// Mitsubishi GX Works2 project: plc_torque1   PLC: FX3U/FX3UC

PROGRAM MAIN
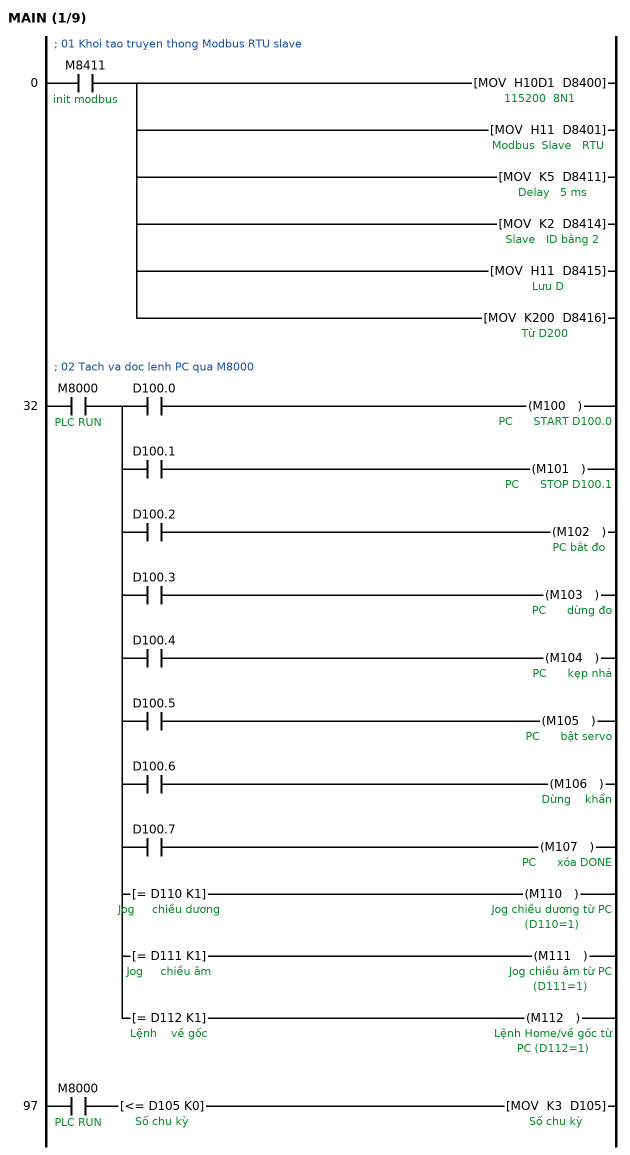
; 01 Khoi tao truyen thong Modbus RTU slave
0     LD      M8411  ; init modbus
      MOV     H10D1 D8400  ; 115200  8N1
      MOV     H11 D8401  ; Modbus  Slave   RTU
      MOV     K5 D8411  ; Delay   5 ms
      MOV     K2 D8414  ; Slave   ID bằng 2
      MOV     H11 D8415  ; Lưu D
      MOV     K200 D8416  ; Từ D200
; 02 Tach va doc lenh PC qua M8000
32    LD      M8000  ; PLC RUN
      MPS
      AND     D100.0
      OUT     M100  ; PC      START D100.0
      MRD
      AND     D100.1
      OUT     M101  ; PC      STOP D100.1
      MRD
      AND     D100.2
      OUT     M102  ; PC bắt đo
      MRD
      AND     D100.3
      OUT     M103  ; PC      dừng đo
      MRD
      AND     D100.4
      OUT     M104  ; PC      kẹp nhả
      MRD
      AND     D100.5
      OUT     M105  ; PC      bật servo
      MRD
      AND     D100.6
      OUT     M106  ; Dừng    khẩn
      MRD
      AND     D100.7
      OUT     M107  ; PC      xóa DONE
      MRD
      LD=     D110 K1  ; Jog     chiều dương
      ANB
      OUT     M110  ; Jog chiều dương từ PC (D110=1)
      MRD
      LD=     D111 K1  ; Jog     chiều âm
      ANB
      OUT     M111  ; Jog chiều âm từ PC (D111=1)
      MPP
      LD=     D112 K1  ; Lệnh    về gốc
      ANB
      OUT     M112  ; Lệnh Home/về gốc từ PC (D112=1)
97    LD      M8000  ; PLC RUN
      AND<=   D105 K0  ; Số chu kỳ
      MOV     K3 D105
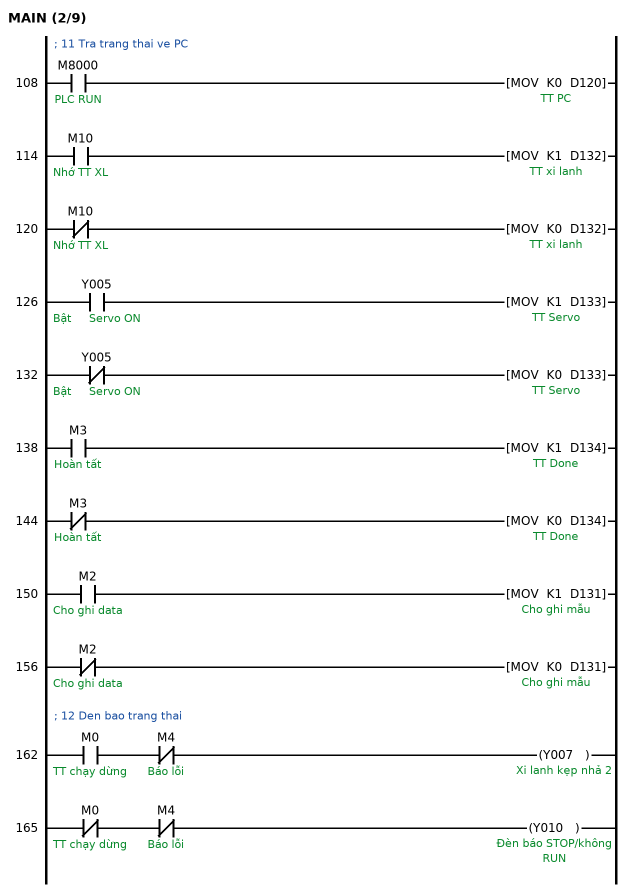
; 11 Tra trang thai ve PC
108   LD      M8000  ; PLC RUN
      MOV     K0 D120  ; TT PC
114   LD      M10  ; Nhớ TT XL
      MOV     K1 D132  ; TT xi lanh
120   LDI     M10  ; Nhớ TT XL
      MOV     K0 D132
126   LD      Y005  ; Bật     Servo ON
      MOV     K1 D133  ; TT Servo
132   LDI     Y005  ; Bật     Servo ON
      MOV     K0 D133
138   LD      M3  ; Hoàn tất
      MOV     K1 D134  ; TT Done
144   LDI     M3  ; Hoàn tất
      MOV     K0 D134
150   LD      M2  ; Cho ghi data
      MOV     K1 D131  ; Cho ghi mẫu
156   LDI     M2  ; Cho ghi data
      MOV     K0 D131
; 12 Den bao trang thai
162   LD      M0  ; TT chạy dừng
      ANI     M4  ; Báo lỗi
      OUT     Y007  ; Xi lanh kẹp nhả 2
165   LDI     M0  ; TT chạy dừng
      ANI     M4  ; Báo lỗi
      OUT     Y010  ; Đèn báo STOP/không RUN
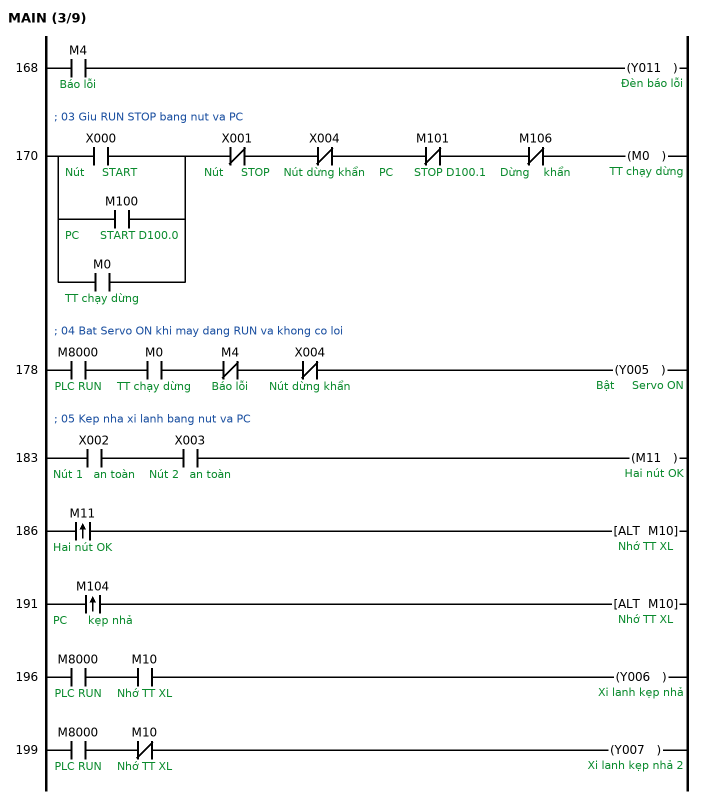
168   LD      M4  ; Báo lỗi
      OUT     Y011  ; Đèn báo lỗi
; 03 Giu RUN STOP bang nut va PC
170   LD      X000  ; Nút     START
      OR      M100  ; PC      START D100.0
      OR      M0  ; TT chạy dừng
      ANI     X001  ; Nút     STOP
      ANI     X004  ; Nút dừng khẩn
      ANI     M101  ; PC      STOP D100.1
      ANI     M106  ; Dừng    khẩn
      OUT     M0  ; TT chạy dừng
; 04 Bat Servo ON khi may dang RUN va khong co loi
178   LD      M8000  ; PLC RUN
      AND     M0  ; TT chạy dừng
      ANI     M4  ; Báo lỗi
      ANI     X004  ; Nút dừng khẩn
      OUT     Y005  ; Bật     Servo ON
; 05 Kep nha xi lanh bang nut va PC
183   LD      X002  ; Nút 1   an toàn
      AND     X003  ; Nút 2   an toàn
      OUT     M11  ; Hai nút OK
186   LDP     M11  ; Hai nút OK
      ALT     M10
191   LDP     M104  ; PC      kẹp nhả
      ALT     M10
196   LD      M8000  ; PLC RUN
      AND     M10  ; Nhớ TT XL
      OUT     Y006  ; Xi lanh kẹp nhả
199   LD      M8000  ; PLC RUN
      ANI     M10  ; Nhớ TT XL
      OUT     Y007  ; Xi lanh kẹp nhả 2
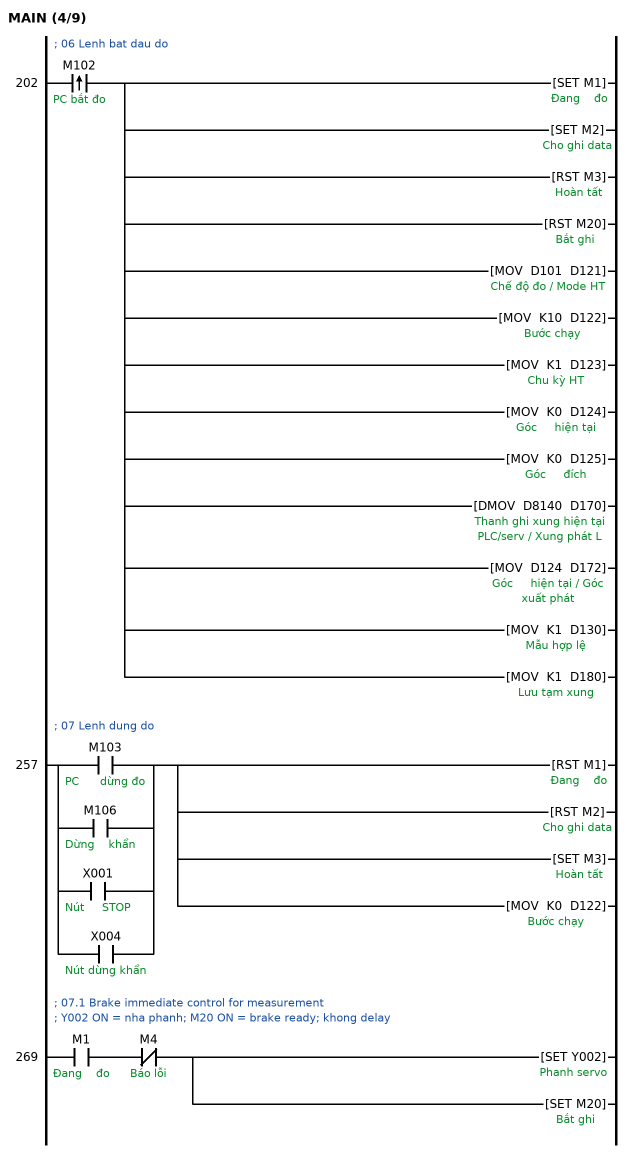
; 06 Lenh bat dau do
202   LDP     M102  ; PC bắt đo
      SET     M1  ; Đang    đo
      SET     M2  ; Cho ghi data
      RST     M3  ; Hoàn tất
      RST     M20  ; Bắt ghi
      MOV     D101 D121  ; Chế độ đo / Mode HT
      MOV     K10 D122  ; Bước chạy
      MOV     K1 D123  ; Chu kỳ HT
      MOV     K0 D124  ; Góc     hiện tại
      MOV     K0 D125  ; Góc     đích
      DMOV    D8140 D170  ; Thanh ghi xung hiện tại PLC/serv / Xung phát L
      MOV     D124 D172  ; Góc xuất phát
      MOV     K1 D130  ; Mẫu hợp lệ
      MOV     K1 D180  ; Lưu tạm xung
; 07 Lenh dung do
257   LD      M103  ; PC      dừng đo
      OR      M106  ; Dừng    khẩn
      OR      X001  ; Nút     STOP
      OR      X004  ; Nút dừng khẩn
      RST     M1  ; Đang    đo
      RST     M2  ; Cho ghi data
      SET     M3  ; Hoàn tất
      MOV     K0 D122
; 07.1 Brake immediate control for measurement
; Y002 ON = nha phanh; M20 ON = brake ready; khong delay
269   LD      M1  ; Đang    đo
      ANI     M4  ; Báo lỗi
      SET     Y002  ; Phanh servo
      SET     M20  ; Bắt ghi
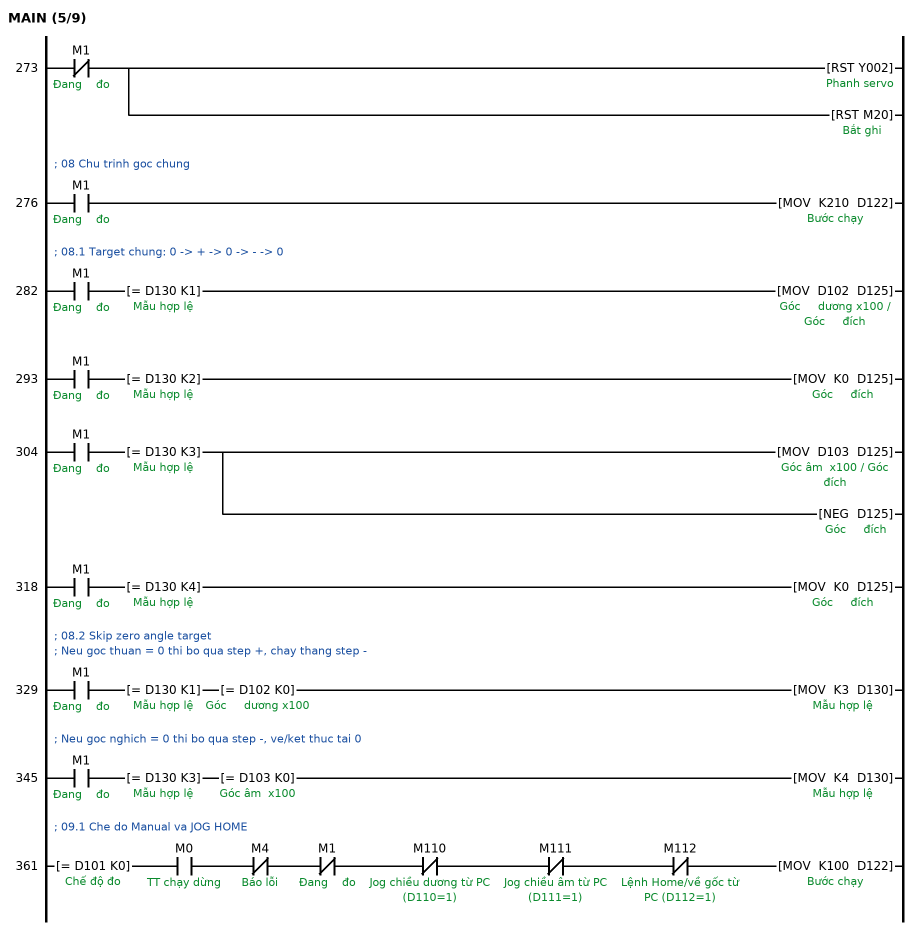
273   LDI     M1  ; Đang    đo
      RST     Y002  ; Phanh servo
      RST     M20  ; Bắt ghi
; 08 Chu trinh goc chung
276   LD      M1  ; Đang    đo
      MOV     K210 D122
; 08.1 Target chung: 0 -> + -> 0 -> - -> 0
282   LD      M1  ; Đang    đo
      AND=    D130 K1  ; Mẫu hợp lệ
      MOV     D102 D125  ; Góc     dương x100
293   LD      M1  ; Đang    đo
      AND=    D130 K2  ; Mẫu hợp lệ
      MOV     K0 D125
304   LD      M1  ; Đang    đo
      AND=    D130 K3  ; Mẫu hợp lệ
      MOV     D103 D125  ; Góc âm  x100
      NEG     D125
318   LD      M1  ; Đang    đo
      AND=    D130 K4  ; Mẫu hợp lệ
      MOV     K0 D125
; 08.2 Skip zero angle target
; Neu goc thuan = 0 thi bo qua step +, chay thang step -
329   LD      M1  ; Đang    đo
      AND=    D130 K1  ; Mẫu hợp lệ
      AND=    D102 K0  ; Góc     dương x100
      MOV     K3 D130
; Neu goc nghich = 0 thi bo qua step -, ve/ket thuc tai 0
345   LD      M1  ; Đang    đo
      AND=    D130 K3  ; Mẫu hợp lệ
      AND=    D103 K0  ; Góc âm  x100
      MOV     K4 D130
; 09.1 Che do Manual va JOG HOME
361   LD=     D101 K0  ; Chế độ đo
      AND     M0  ; TT chạy dừng
      ANI     M4  ; Báo lỗi
      ANI     M1  ; Đang    đo
      ANI     M110  ; Jog chiều dương từ PC (D110=1)
      ANI     M111  ; Jog chiều âm từ PC (D111=1)
      ANI     M112  ; Lệnh Home/về gốc từ PC (D112=1)
      MOV     K100 D122
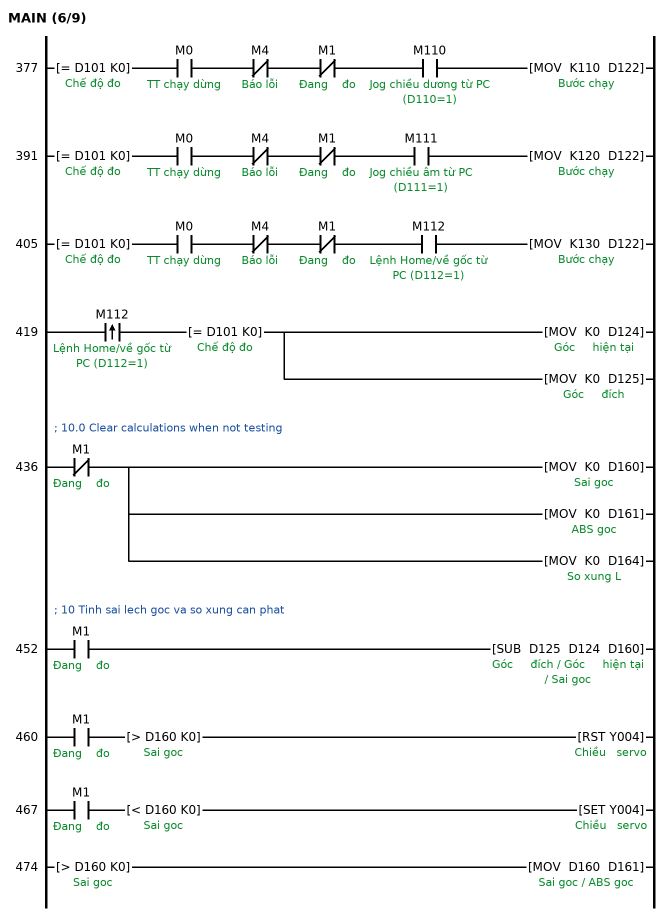
377   LD=     D101 K0  ; Chế độ đo
      AND     M0  ; TT chạy dừng
      ANI     M4  ; Báo lỗi
      ANI     M1  ; Đang    đo
      AND     M110  ; Jog chiều dương từ PC (D110=1)
      MOV     K110 D122
391   LD=     D101 K0  ; Chế độ đo
      AND     M0  ; TT chạy dừng
      ANI     M4  ; Báo lỗi
      ANI     M1  ; Đang    đo
      AND     M111  ; Jog chiều âm từ PC (D111=1)
      MOV     K120 D122
405   LD=     D101 K0  ; Chế độ đo
      AND     M0  ; TT chạy dừng
      ANI     M4  ; Báo lỗi
      ANI     M1  ; Đang    đo
      AND     M112  ; Lệnh Home/về gốc từ PC (D112=1)
      MOV     K130 D122
419   LDP     M112  ; Lệnh Home/về gốc từ PC (D112=1)
      AND=    D101 K0  ; Chế độ đo
      MOV     K0 D124
      MOV     K0 D125
; 10.0 Clear calculations when not testing
436   LDI     M1  ; Đang    đo
      MOV     K0 D160  ; Sai goc
      MOV     K0 D161  ; ABS goc
      MOV     K0 D164  ; So xung L
; 10 Tinh sai lech goc va so xung can phat
452   LD      M1  ; Đang    đo
      SUB     D125 D124 D160
460   LD      M1  ; Đang    đo
      AND>    D160 K0  ; Sai goc
      RST     Y004  ; Chiều   servo
467   LD      M1  ; Đang    đo
      AND<    D160 K0  ; Sai goc
      SET     Y004  ; Chiều   servo
474   LD>     D160 K0  ; Sai goc
      MOV     D160 D161
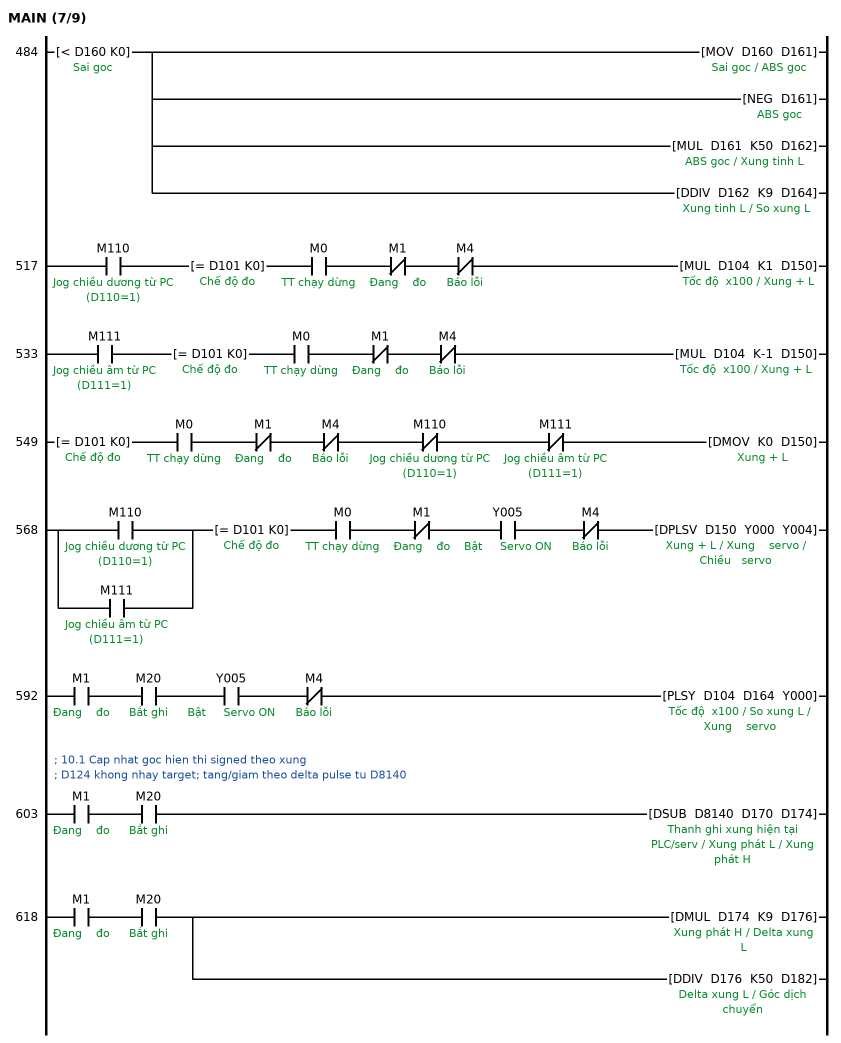
484   LD<     D160 K0  ; Sai goc
      MOV     D160 D161
      NEG     D161
      MUL     D161 K50 D162  ; Xung tinh L
      DDIV    D162 K9 D164
517   LD      M110  ; Jog chiều dương từ PC (D110=1)
      AND=    D101 K0  ; Chế độ đo
      AND     M0  ; TT chạy dừng
      ANI     M1  ; Đang    đo
      ANI     M4  ; Báo lỗi
      MUL     D104 K1 D150  ; Tốc độ  x100 / Xung + L
533   LD      M111  ; Jog chiều âm từ PC (D111=1)
      AND=    D101 K0  ; Chế độ đo
      AND     M0  ; TT chạy dừng
      ANI     M1  ; Đang    đo
      ANI     M4  ; Báo lỗi
      MUL     D104 K-1 D150
549   LD=     D101 K0  ; Chế độ đo
      AND     M0  ; TT chạy dừng
      ANI     M1  ; Đang    đo
      ANI     M4  ; Báo lỗi
      ANI     M110  ; Jog chiều dương từ PC (D110=1)
      ANI     M111  ; Jog chiều âm từ PC (D111=1)
      DMOV    K0 D150
568   LD      M110  ; Jog chiều dương từ PC (D110=1)
      OR      M111  ; Jog chiều âm từ PC (D111=1)
      AND=    D101 K0  ; Chế độ đo
      AND     M0  ; TT chạy dừng
      ANI     M1  ; Đang    đo
      AND     Y005  ; Bật     Servo ON
      ANI     M4  ; Báo lỗi
      DPLSV   D150 Y000 Y004  ; Xung    servo
592   LD      M1  ; Đang    đo
      AND     M20  ; Bắt ghi
      AND     Y005  ; Bật     Servo ON
      ANI     M4  ; Báo lỗi
      PLSY    D104 D164 Y000  ; Tốc độ  x100 / So xung L / Xung    servo
; 10.1 Cap nhat goc hien thi signed theo xung
; D124 khong nhay target; tang/giam theo delta pulse tu D8140
603   LD      M1  ; Đang    đo
      AND     M20  ; Bắt ghi
      DSUB    D8140 D170 D174  ; Xung phát H
618   LD      M1  ; Đang    đo
      AND     M20  ; Bắt ghi
      DMUL    D174 K9 D176  ; Delta xung L
      DDIV    D176 K50 D182  ; Góc dịch chuyển
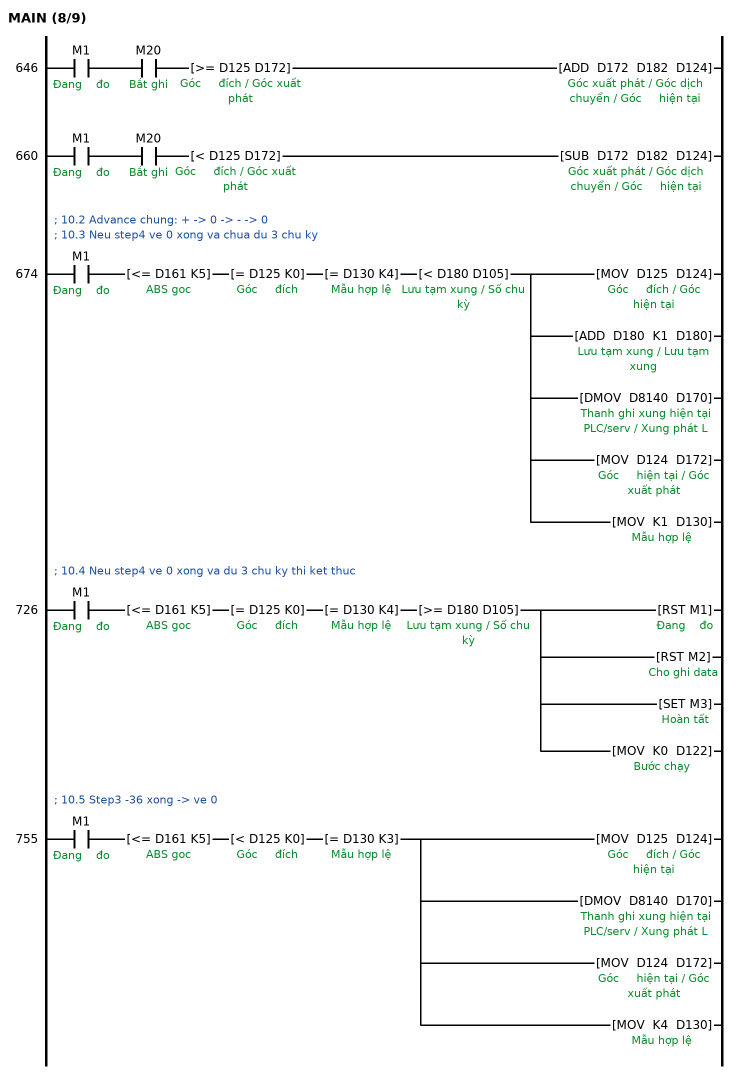
646   LD      M1  ; Đang    đo
      AND     M20  ; Bắt ghi
      AND>=   D125 D172  ; Góc     đích / Góc xuất phát
      ADD     D172 D182 D124
660   LD      M1  ; Đang    đo
      AND     M20  ; Bắt ghi
      AND<    D125 D172  ; Góc     đích / Góc xuất phát
      SUB     D172 D182 D124
; 10.2 Advance chung: + -> 0 -> - -> 0
; 10.3 Neu step4 ve 0 xong va chua du 3 chu ky
674   LD      M1  ; Đang    đo
      AND<=   D161 K5  ; ABS goc
      AND=    D125 K0  ; Góc     đích
      AND=    D130 K4  ; Mẫu hợp lệ
      AND<    D180 D105  ; Lưu tạm xung / Số chu kỳ
      MOV     D125 D124
      ADD     D180 K1 D180
      DMOV    D8140 D170
      MOV     D124 D172
      MOV     K1 D130
; 10.4 Neu step4 ve 0 xong va du 3 chu ky thi ket thuc
726   LD      M1  ; Đang    đo
      AND<=   D161 K5  ; ABS goc
      AND=    D125 K0  ; Góc     đích
      AND=    D130 K4  ; Mẫu hợp lệ
      AND>=   D180 D105  ; Lưu tạm xung / Số chu kỳ
      RST     M1  ; Đang    đo
      RST     M2  ; Cho ghi data
      SET     M3  ; Hoàn tất
      MOV     K0 D122
; 10.5 Step3 -36 xong -> ve 0
755   LD      M1  ; Đang    đo
      AND<=   D161 K5  ; ABS goc
      AND<    D125 K0  ; Góc     đích
      AND=    D130 K3  ; Mẫu hợp lệ
      MOV     D125 D124
      DMOV    D8140 D170
      MOV     D124 D172
      MOV     K4 D130
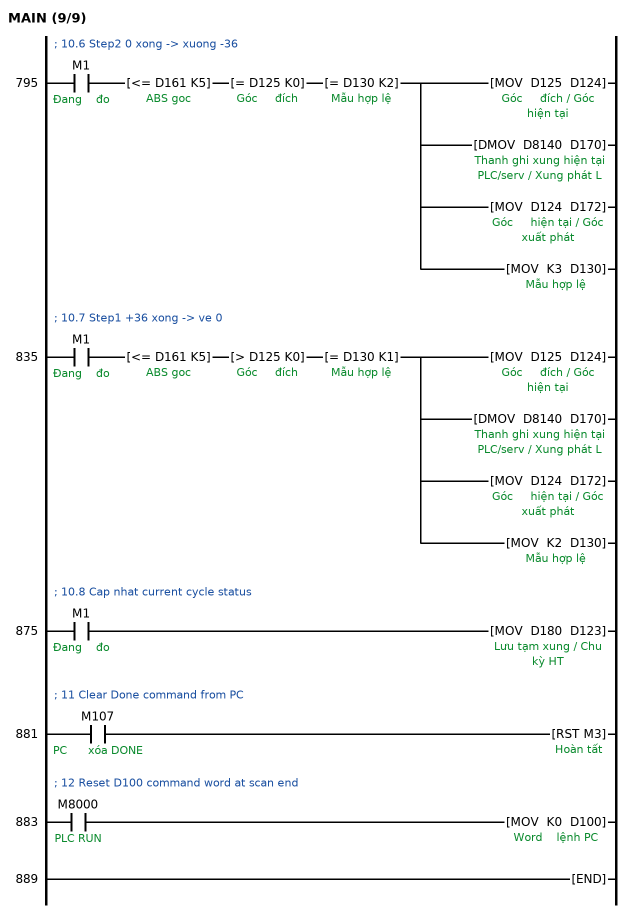
; 10.6 Step2 0 xong -> xuong -36
795   LD      M1  ; Đang    đo
      AND<=   D161 K5  ; ABS goc
      AND=    D125 K0  ; Góc     đích
      AND=    D130 K2  ; Mẫu hợp lệ
      MOV     D125 D124
      DMOV    D8140 D170
      MOV     D124 D172
      MOV     K3 D130
; 10.7 Step1 +36 xong -> ve 0
835   LD      M1  ; Đang    đo
      AND<=   D161 K5  ; ABS goc
      AND>    D125 K0  ; Góc     đích
      AND=    D130 K1  ; Mẫu hợp lệ
      MOV     D125 D124
      DMOV    D8140 D170
      MOV     D124 D172
      MOV     K2 D130
; 10.8 Cap nhat current cycle status
875   LD      M1  ; Đang    đo
      MOV     D180 D123
; 11 Clear Done command from PC
881   LD      M107  ; PC      xóa DONE
      RST     M3  ; Hoàn tất
; 12 Reset D100 command word at scan end
883   LD      M8000  ; PLC RUN
      MOV     K0 D100  ; Word    lệnh PC
889   END
END_PROGRAM

// device comments not shown above
M12  ; Xung 2 nút
M13  ; PC kẹp nhả
M21  ; Dừng ghi
M30  ; SV đang chạy
M31  ; SV chạy xong
M32  ; SV chiều +
M33  ; SV chiều -
D106  ; Vùng    lấy mẫu
D107  ; Chọn    loại SP
D108  ; Loại    đo momen
D109  ; Reset   lỗi PC
D126  ; Tốc độ HT
D127  ; VT servo L
D128  ; VT servo H
D129  ; Mã lỗi  PLC
D135  ; Số mẫu
D151  ; Xung + H
D152  ; Xung - L
D153  ; Xung - H
D154  ; Tốc xung L
D155  ; Tốc xung H
D156  ; Góc min OK
D157  ; Góc max OK
D158  ; TG bước
D163  ; Xung tinh H
D165  ; So xung H
